{attribute addProperty BoxType "EK1100-0000-0018"}
{attribute addProperty Id "Beckhoff_AX8yxxEK1122Beckhoff_AX8yxxEK1122_029BE14F1008126A_0001_AX8108_0000_0041AX8108_A2FEB36A47259A_0002_AX8108_0000_0100AX8108_D97ACBDE40851A_0003_AX8108_0000_0101AX8108_D97ACBDE40851A_0004_AX8108_0000_0102AX8108_3F1F35B340851A_0005_AX8108_0000_0103AX8108_3F1F35B340851A_0006_AX8108_0000_0104AX8108_3F1F35B340851A_0007_AX8108_0010_0102AX8108_3F1F35B340851A_0008_AX8108_0010_0103AX8108_3F1F35B340851A_0009_AX8108_0010_0104AX8108_3F1F35B340851A_0010_AX8108_0100_0101AX8108_6A10D9BF58473A_0011_AX8108_0100_0102AX8108_8C7527D258473A_0012_AX8108_0100_0103AX8108_8C7527D258473A_0013_AX8108_0100_0104AX8108_8C7527D258473A_0014_AX8108_0110_0102AX8108_8C7527D258473A_0015_AX8108_0110_0103AX8108_8C7527D258473A_0016_AX8108_0110_0104AX8108_8C7527D258473A_0017_AX8108_0200_0103AX8108_8C7527D258473A_0018_AX8108_0200_0104AX8108_8C7527D258473A_0019_AX8108_0210_0103AX8108_8C7527D258473A_0020_AX8108_0210_0104AX8108_8C7527D258473A_0021_AX8118_0000_0041AX8118_A2FEB36A47259A_0022_AX8118_0000_0100AX8118_D97ACBDE40851A_0023_AX8118_0000_0101AX8118_D97ACBDE40851A_0024_AX8118_0000_0102AX8118_3F1F35B340851A_0025_AX8118_0000_0103AX8118_3F1F35B340851A_0026_AX8118_0000_0104AX8118_3F1F35B340851A_0027_AX8118_0010_0102AX8118_3F1F35B340851A_0028_AX8118_0010_0103AX8118_3F1F35B340851A_0029_AX8118_0010_0104AX8118_3F1F35B340851A_0030_AX8118_0100_0101AX8118_6A10D9BF58473A_0031_AX8118_0100_0102AX8118_8C7527D258473A_0032_AX8118_0100_0103AX8118_8C7527D258473A_0033_AX8118_0100_0104AX8118_8C7527D258473A_0034_AX8118_0110_0102AX8118_8C7527D258473A_0035_AX8118_0110_0103AX8118_8C7527D258473A_0036_AX8118_0110_0104AX8118_8C7527D258473A_0037_AX8118_0200_0103AX8118_8C7527D258473A_0038_AX8118_0200_0104AX8118_8C7527D258473A_0039_AX8118_0210_0103AX8118_8C7527D258473A_0040_AX8118_0210_0104AX8118_8C7527D258473A_0041_AX8206_0000_0041AX8206_D62D632572090A_0042_AX8206_0000_0100AX8206_D4C3F58959274A_0043_AX8206_0000_0101AX8206_D4C3F58959274A_0044_AX8206_0000_0102AX8206_DA6659A959274A_0045_AX8206_0000_0103AX8206_DA6659A959274A_0046_AX8206_0000_0104AX8206_DA6659A959274A_0047_AX8206_0010_0102AX8206_DA6659A959274A_0048_AX8206_0010_0103AX8206_DA6659A959274A_0049_AX8206_0010_0104AX8206_DA6659A959274A_0050_AX8206_0100_0101AX8206_8FDEBF0476896A_0051_AX8206_0100_0102AX8206_817B132476896A_0052_AX8206_0100_0103AX8206_817B132476896A_0053_AX8206_0100_0104AX8206_817B132476896A_0054_AX8206_0110_0102AX8206_817B132476896A_0055_AX8206_0110_0103AX8206_817B132476896A_0056_AX8206_0110_0104AX8206_817B132476896A_0057_AX8206_0200_0103AX8206_817B132476896A_0058_AX8206_0200_0104AX8206_817B132476896A_0059_AX8206_0210_0103AX8206_817B132476896A_0060_AX8206_0210_0104AX8206_817B132476896"}
{attribute addProperty CRC "3929363410"}
{attribute addProperty SizeInBites "35232"}
{attribute addProperty SizeInBytes "4404"}
TYPE Beckhoff_AX8yxx_EA3553D2 EXTENDS EK1100_179A0949 :
STRUCT
	{attribute addProperty Name "Beckhoff_AX8yxxEK1122"}
	Beckhoff_AX8yxxEK1122 : Beckhoff_AX8yxxEK1122_029BE14F;
	{attribute addProperty Name "A_0001_AX8108_0000_0041"}
	A_0001_AX8108_0000_0041 : AX8108_A2FEB36A;
	{attribute addProperty Name "A_0002_AX8108_0000_0100"}
	A_0002_AX8108_0000_0100 : AX8108_D97ACBDE;
	{attribute addProperty Name "A_0003_AX8108_0000_0101"}
	A_0003_AX8108_0000_0101 : AX8108_D97ACBDE;
	{attribute addProperty Name "A_0004_AX8108_0000_0102"}
	A_0004_AX8108_0000_0102 : AX8108_3F1F35B3;
	{attribute addProperty Name "A_0005_AX8108_0000_0103"}
	A_0005_AX8108_0000_0103 : AX8108_3F1F35B3;
	{attribute addProperty Name "A_0006_AX8108_0000_0104"}
	A_0006_AX8108_0000_0104 : AX8108_3F1F35B3;
	{attribute addProperty Name "A_0007_AX8108_0010_0102"}
	A_0007_AX8108_0010_0102 : AX8108_3F1F35B3;
	{attribute addProperty Name "A_0008_AX8108_0010_0103"}
	A_0008_AX8108_0010_0103 : AX8108_3F1F35B3;
	{attribute addProperty Name "A_0009_AX8108_0010_0104"}
	A_0009_AX8108_0010_0104 : AX8108_3F1F35B3;
	{attribute addProperty Name "A_0010_AX8108_0100_0101"}
	A_0010_AX8108_0100_0101 : AX8108_6A10D9BF;
	{attribute addProperty Name "A_0011_AX8108_0100_0102"}
	A_0011_AX8108_0100_0102 : AX8108_8C7527D2;
	{attribute addProperty Name "A_0012_AX8108_0100_0103"}
	A_0012_AX8108_0100_0103 : AX8108_8C7527D2;
	{attribute addProperty Name "A_0013_AX8108_0100_0104"}
	A_0013_AX8108_0100_0104 : AX8108_8C7527D2;
	{attribute addProperty Name "A_0014_AX8108_0110_0102"}
	A_0014_AX8108_0110_0102 : AX8108_8C7527D2;
	{attribute addProperty Name "A_0015_AX8108_0110_0103"}
	A_0015_AX8108_0110_0103 : AX8108_8C7527D2;
	{attribute addProperty Name "A_0016_AX8108_0110_0104"}
	A_0016_AX8108_0110_0104 : AX8108_8C7527D2;
	{attribute addProperty Name "A_0017_AX8108_0200_0103"}
	A_0017_AX8108_0200_0103 : AX8108_8C7527D2;
	{attribute addProperty Name "A_0018_AX8108_0200_0104"}
	A_0018_AX8108_0200_0104 : AX8108_8C7527D2;
	{attribute addProperty Name "A_0019_AX8108_0210_0103"}
	A_0019_AX8108_0210_0103 : AX8108_8C7527D2;
	{attribute addProperty Name "A_0020_AX8108_0210_0104"}
	A_0020_AX8108_0210_0104 : AX8108_8C7527D2;
	{attribute addProperty Name "A_0021_AX8118_0000_0041"}
	A_0021_AX8118_0000_0041 : AX8118_A2FEB36A;
	{attribute addProperty Name "A_0022_AX8118_0000_0100"}
	A_0022_AX8118_0000_0100 : AX8118_D97ACBDE;
	{attribute addProperty Name "A_0023_AX8118_0000_0101"}
	A_0023_AX8118_0000_0101 : AX8118_D97ACBDE;
	{attribute addProperty Name "A_0024_AX8118_0000_0102"}
	A_0024_AX8118_0000_0102 : AX8118_3F1F35B3;
	{attribute addProperty Name "A_0025_AX8118_0000_0103"}
	A_0025_AX8118_0000_0103 : AX8118_3F1F35B3;
	{attribute addProperty Name "A_0026_AX8118_0000_0104"}
	A_0026_AX8118_0000_0104 : AX8118_3F1F35B3;
	{attribute addProperty Name "A_0027_AX8118_0010_0102"}
	A_0027_AX8118_0010_0102 : AX8118_3F1F35B3;
	{attribute addProperty Name "A_0028_AX8118_0010_0103"}
	A_0028_AX8118_0010_0103 : AX8118_3F1F35B3;
	{attribute addProperty Name "A_0029_AX8118_0010_0104"}
	A_0029_AX8118_0010_0104 : AX8118_3F1F35B3;
	{attribute addProperty Name "A_0030_AX8118_0100_0101"}
	A_0030_AX8118_0100_0101 : AX8118_6A10D9BF;
	{attribute addProperty Name "A_0031_AX8118_0100_0102"}
	A_0031_AX8118_0100_0102 : AX8118_8C7527D2;
	{attribute addProperty Name "A_0032_AX8118_0100_0103"}
	A_0032_AX8118_0100_0103 : AX8118_8C7527D2;
	{attribute addProperty Name "A_0033_AX8118_0100_0104"}
	A_0033_AX8118_0100_0104 : AX8118_8C7527D2;
	{attribute addProperty Name "A_0034_AX8118_0110_0102"}
	A_0034_AX8118_0110_0102 : AX8118_8C7527D2;
	{attribute addProperty Name "A_0035_AX8118_0110_0103"}
	A_0035_AX8118_0110_0103 : AX8118_8C7527D2;
	{attribute addProperty Name "A_0036_AX8118_0110_0104"}
	A_0036_AX8118_0110_0104 : AX8118_8C7527D2;
	{attribute addProperty Name "A_0037_AX8118_0200_0103"}
	A_0037_AX8118_0200_0103 : AX8118_8C7527D2;
	{attribute addProperty Name "A_0038_AX8118_0200_0104"}
	A_0038_AX8118_0200_0104 : AX8118_8C7527D2;
	{attribute addProperty Name "A_0039_AX8118_0210_0103"}
	A_0039_AX8118_0210_0103 : AX8118_8C7527D2;
	{attribute addProperty Name "A_0040_AX8118_0210_0104"}
	A_0040_AX8118_0210_0104 : AX8118_8C7527D2;
	{attribute addProperty Name "A_0041_AX8206_0000_0041"}
	A_0041_AX8206_0000_0041 : AX8206_D62D6325;
	{attribute addProperty Name "A_0042_AX8206_0000_0100"}
	A_0042_AX8206_0000_0100 : AX8206_D4C3F589;
	{attribute addProperty Name "A_0043_AX8206_0000_0101"}
	A_0043_AX8206_0000_0101 : AX8206_D4C3F589;
	{attribute addProperty Name "A_0044_AX8206_0000_0102"}
	A_0044_AX8206_0000_0102 : AX8206_DA6659A9;
	{attribute addProperty Name "A_0045_AX8206_0000_0103"}
	A_0045_AX8206_0000_0103 : AX8206_DA6659A9;
	{attribute addProperty Name "A_0046_AX8206_0000_0104"}
	A_0046_AX8206_0000_0104 : AX8206_DA6659A9;
	{attribute addProperty Name "A_0047_AX8206_0010_0102"}
	A_0047_AX8206_0010_0102 : AX8206_DA6659A9;
	{attribute addProperty Name "A_0048_AX8206_0010_0103"}
	A_0048_AX8206_0010_0103 : AX8206_DA6659A9;
	{attribute addProperty Name "A_0049_AX8206_0010_0104"}
	A_0049_AX8206_0010_0104 : AX8206_DA6659A9;
	{attribute addProperty Name "A_0050_AX8206_0100_0101"}
	A_0050_AX8206_0100_0101 : AX8206_8FDEBF04;
	{attribute addProperty Name "A_0051_AX8206_0100_0102"}
	A_0051_AX8206_0100_0102 : AX8206_817B1324;
	{attribute addProperty Name "A_0052_AX8206_0100_0103"}
	A_0052_AX8206_0100_0103 : AX8206_817B1324;
	{attribute addProperty Name "A_0053_AX8206_0100_0104"}
	A_0053_AX8206_0100_0104 : AX8206_817B1324;
	{attribute addProperty Name "A_0054_AX8206_0110_0102"}
	A_0054_AX8206_0110_0102 : AX8206_817B1324;
	{attribute addProperty Name "A_0055_AX8206_0110_0103"}
	A_0055_AX8206_0110_0103 : AX8206_817B1324;
	{attribute addProperty Name "A_0056_AX8206_0110_0104"}
	A_0056_AX8206_0110_0104 : AX8206_817B1324;
	{attribute addProperty Name "A_0057_AX8206_0200_0103"}
	A_0057_AX8206_0200_0103 : AX8206_817B1324;
	{attribute addProperty Name "A_0058_AX8206_0200_0104"}
	A_0058_AX8206_0200_0104 : AX8206_817B1324;
	{attribute addProperty Name "A_0059_AX8206_0210_0103"}
	A_0059_AX8206_0210_0103 : AX8206_817B1324;
	{attribute addProperty Name "A_0060_AX8206_0210_0104"}
	A_0060_AX8206_0210_0104 : AX8206_817B1324;
END_STRUCT
END_TYPE

(* stored: Version 1.2.0.0, ProductVersion 3.1.4024.9
   DUT Beckhoff_AX8yxx_EA3553D2: Id {7acdbd7d-76db-437b-bdb9-f14698689f5c} *)
